INTERFACE IReadOnlyByteList EXTENDS IPointerCollection

METHOD Get : BYTE
VAR_INPUT
	index : DINT;
END_VAR
END_METHOD

END_INTERFACE

(* stored: Version 1.1.0.1
   Itf IReadOnlyByteList: Id {a843c369-9e00-00a1-32fa-d03c5ab85265}
   Method Get: Id {27925820-f345-0e43-1a3c-84ba47105d29} *)
